(* Logix 5000 project; controller WAGO_765_1504_Sample vendor 1 type 14 code 196 rev 32.14; software revision 32.03 *)

TASK MainTask (continuous, watchdog 500 ms) : MainProgram

MODULES
   Local : vendor 1 type 14 code 196 (5069 0, rev 32.14)
      WAGO_DIO_1504 : vendor 40 type 12 code 1504 (Ethernet 192.168.2.100, rev 1.1, StandardDataDriven RPI 20 ms)
END_MODULES

ADD_ON_INSTRUCTION WAGO_765_1504   (* revision 1.1, vendor WAGO *)
// 765-1504/100-000 AOI, Exclusive Owner Connection Type
// Revision note:
// ModuleConfig.DIO_Process_Data_Layout can be 1 or 0. DO data release is now written to
// Help:
// The WAGO_765_1504 instruction normalizes data received from a WAGO 750-1504/100-000 DIO EIP Adapter. 765-1504/100-000 must be Exclusive Owner (with config).
// This AOI requires ModuleConfig, ModuleInput, and ModuleOutput. These data types are from the EDS file, so do not create these data types--they should already be there if you have the device added.
// ModuleConfig is of type _0028:765_15040100_0000_419E4C60:C:0. This data type allows for configuration of the 765-1504 EIP Adapter.
// ModuleInput is of type _0028:765_15040100_0000_85D36DB4:I:0
// ModuleOutput is of type _0028:765_15040100_0000_AAB94180:O:0
// These data types are from the connection class and should be easily assignable.
// Each port has a pin 2 and pin 4 for input/output data. The DIO configuration is done through the ModuleConfig within the Network Variables. The AOI will break out each pin into individual BOOLs to ease referencing.
// Consult the WAGO 765-1504/100-000 Product Manual for further information about the WAGO I/O System Field DIO EIP Adapter.
VAR_IN_OUT
   ModuleConfig : _0028:765_15040100_0000_419E4C60:C:0; {required}
   ModuleInputs : _0028:765_15040100_0000_85D36DB4:I:0; {required}
   ModuleOutputs : _0028:765_15040100_0000_AAB94180:O:0; {required}
END_VAR
VAR_OUTPUT
   X01_Pin4_Input : BOOL; {access None, visible}
END_VAR
VAR_INPUT
   X01_Pin4_Output : BOOL; {access None, visible}
END_VAR
VAR_OUTPUT
   X01_Pin2_Input : BOOL; {access None, visible}
END_VAR
VAR_INPUT
   X01_Pin2_Output : BOOL; {access None, visible}
END_VAR
VAR_OUTPUT
   X02_Pin4_Input : BOOL; {access None, visible}
END_VAR
VAR_INPUT
   X02_Pin4_Output : BOOL; {access None, visible}
END_VAR
VAR_OUTPUT
   X02_Pin2_Input : BOOL; {access None, visible}
END_VAR
VAR_INPUT
   X02_Pin2_Output : BOOL; {access None, visible}
END_VAR
VAR_OUTPUT
   X03_Pin4_Input : BOOL; {access None, visible}
END_VAR
VAR_INPUT
   X03_Pin4_Output : BOOL; {access None, visible}
END_VAR
VAR_OUTPUT
   X03_Pin2_Input : BOOL; {access None, visible}
END_VAR
VAR_INPUT
   X03_Pin2_Output : BOOL; {access None, visible}
END_VAR
VAR_OUTPUT
   X04_Pin4_Input : BOOL; {access None, visible}
END_VAR
VAR_INPUT
   X04_Pin4_Output : BOOL; {access None, visible}
END_VAR
VAR_OUTPUT
   X04_Pin2_Input : BOOL; {access None, visible}
END_VAR
VAR_INPUT
   X04_Pin2_Output : BOOL; {access None, visible}
END_VAR
VAR
   Step : BOOL; {access None}
END_VAR

ROUTINE Logic   (* ladder *)
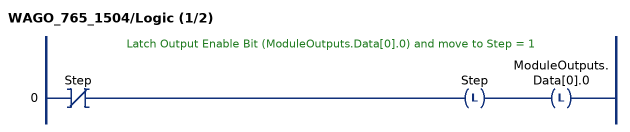
   // Latch Output Enable Bit (ModuleOutputs.Data[0].0) and move to Step = 1
   0: XIO(Step)OTL(Step)OTL(ModuleOutputs.Data[0].0);
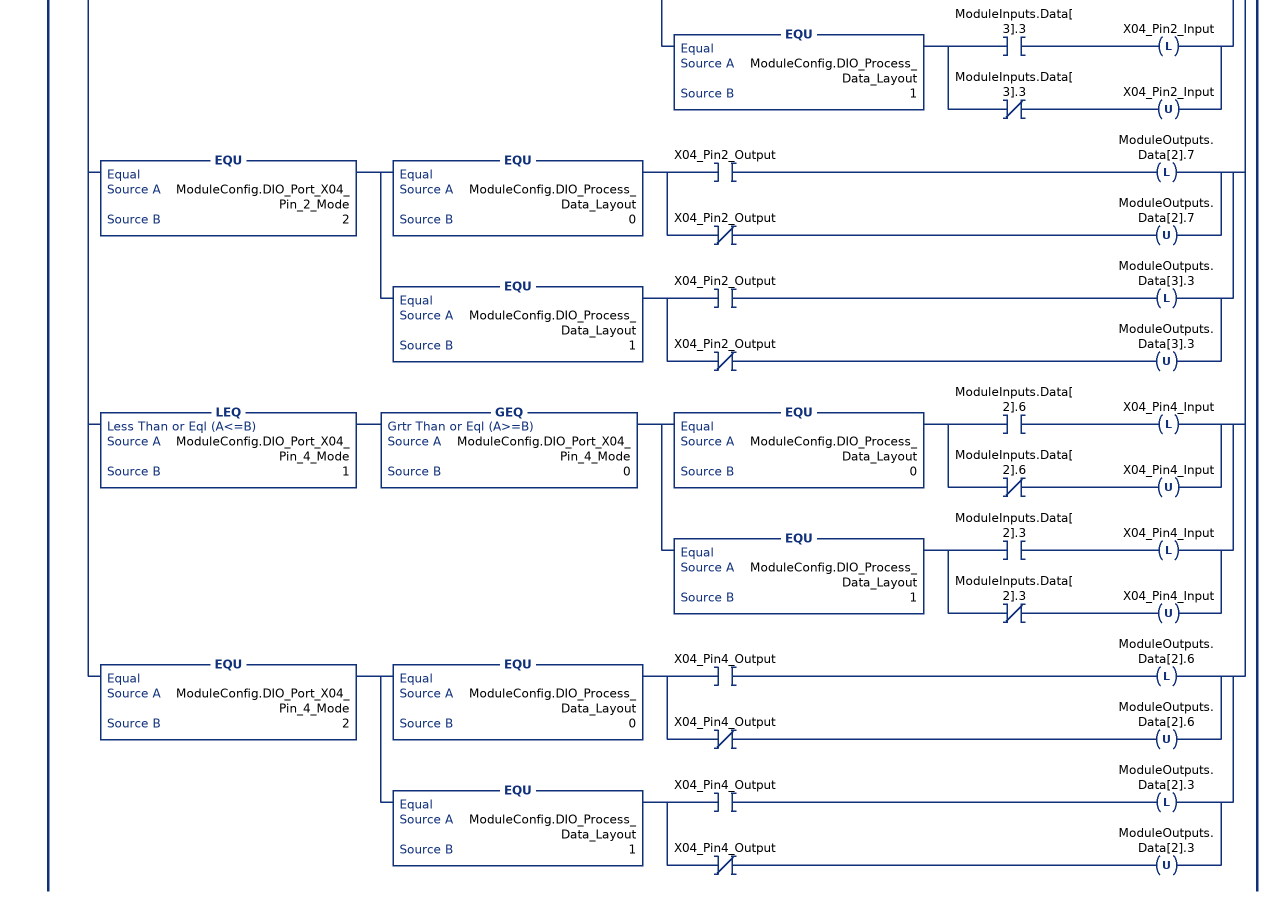
   // Inputs/Outputs read/written are based on ModuleConfig.DIO_Process_Data_Layout.
   1: XIC(Step)[[LEQ(ModuleConfig.DIO_Port_X01_Pin_2_Mode,1) GEQ(ModuleConfig.DIO_Port_X01_Pin_2_Mode,0) [EQU(ModuleConfig.DIO_Process_Data_Layout,0) [XIC(ModuleInputs.Data[2].1) OTL(X01_Pin2_Input) ,XIO(ModuleInputs.Data[2].1) OTU(X01_Pin2_Input) ] ,EQU(ModuleConfig.DIO_Process_Data_Layout,1) [XIC(ModuleInputs.Data[3].0) OTL(X01_Pin2_Input) ,XIO(ModuleInputs.Data[3].0) OTU(X01_Pin2_Input) ] ] ,EQU(ModuleConfig.DIO_Port_X01_Pin_2_Mode,2) [EQU(ModuleConfig.DIO_Process_Data_Layout,0) [XIC(X01_Pin2_Output) OTL(ModuleOutputs.Data[2].1) ,XIO(X01_Pin2_Output) OTU(ModuleOutputs.Data[2].1) ] ,EQU(ModuleConfig.DIO_Process_Data_Layout,1) [XIC(X01_Pin2_Output) OTL(ModuleOutputs.Data[3].0) ,XIO(X01_Pin2_Output) OTU(ModuleOutputs.Data[3].0) ] ] ] ,[LEQ(ModuleConfig.DIO_Port_X01_Pin_4_Mode,1) GEQ(ModuleConfig.DIO_Port_X01_Pin_4_Mode,0) XIC(ModuleInputs.Data[2].0) OTE(X01_Pin4_Input) ,EQU(ModuleConfig.DIO_Port_X01_Pin_4_Mode,2) XIC(X01_Pin4_Output) OTE(ModuleOutputs.Data[2].0) ] ,[LEQ(ModuleConfig.DIO_Port_X02_Pin_2_Mode,1) GEQ(ModuleConfig.DIO_Port_X02_Pin_2_Mode,0) [EQU(ModuleConfig.DIO_Process_Data_Layout,0) [XIC(ModuleInputs.Data[2].3) OTL(X02_Pin2_Input) ,XIO(ModuleInputs.Data[2].3) OTU(X02_Pin2_Input) ] ,EQU(ModuleConfig.DIO_Process_Data_Layout,1) [XIC(ModuleInputs.Data[3].1) OTL(X02_Pin2_Input) ,XIO(ModuleInputs.Data[3].1) OTU(X02_Pin2_Input) ] ] ,EQU(ModuleConfig.DIO_Port_X02_Pin_2_Mode,2) [EQU(ModuleConfig.DIO_Process_Data_Layout,0) [XIC(X02_Pin2_Output) OTL(ModuleOutputs.Data[2].3) ,XIO(X02_Pin2_Output) OTU(ModuleOutputs.Data[2].3) ] ,EQU(ModuleConfig.DIO_Process_Data_Layout,1) [XIC(X02_Pin2_Output) OTL(ModuleOutputs.Data[3].1) ,XIO(X02_Pin2_Output) OTU(ModuleOutputs.Data[3].1) ] ] ] ,[LEQ(ModuleConfig.DIO_Port_X02_Pin_4_Mode,1) GEQ(ModuleConfig.DIO_Port_X02_Pin_4_Mode,0) [EQU(ModuleConfig.DIO_Process_Data_Layout,0) [XIC(ModuleInputs.Data[2].2) OTL(X02_Pin4_Input) ,XIO(ModuleInputs.Data[2].2) OTU(X02_Pin4_Input) ] ,EQU(ModuleConfig.DIO_Process_Data_Layout,1) [XIC(ModuleInputs.Data[2].1) OTL(X02_Pin4_Input) ,XIO(ModuleInputs.Data[2].1) OTU(X02_Pin4_Input) ] ] ,EQU(ModuleConfig.DIO_Port_X02_Pin_4_Mode,2) [EQU(ModuleConfig.DIO_Process_Data_Layout,0) [XIC(X02_Pin4_Output) OTL(ModuleOutputs.Data[2].2) ,XIO(X02_Pin4_Output) OTU(ModuleOutputs.Data[2].2) ] ,EQU(ModuleConfig.DIO_Process_Data_Layout,1) [XIC(X02_Pin4_Output) OTL(ModuleOutputs.Data[2].1) ,XIO(X02_Pin4_Output) OTU(ModuleOutputs.Data[2].1) ] ] ] ,[LEQ(ModuleConfig.DIO_Port_X03_Pin_2_Mode,1) GEQ(ModuleConfig.DIO_Port_X03_Pin_2_Mode,0) [EQU(ModuleConfig.DIO_Process_Data_Layout,0) [XIC(ModuleInputs.Data[2].5) OTL(X03_Pin2_Input) ,XIO(ModuleInputs.Data[2].5) OTU(X03_Pin2_Input) ] ,EQU(ModuleConfig.DIO_Process_Data_Layout,1) [XIC(ModuleInputs.Data[3].2) OTL(X03_Pin2_Input) ,XIO(ModuleInputs.Data[3].2) OTU(X03_Pin2_Input) ] ] ,EQU(ModuleConfig.DIO_Port_X03_Pin_2_Mode,2) [EQU(ModuleConfig.DIO_Process_Data_Layout,0) [XIC(X03_Pin2_Output) OTL(ModuleOutputs.Data[2].5) ,XIO(X03_Pin2_Output) OTU(ModuleOutputs.Data[2].5) ] ,EQU(ModuleConfig.DIO_Process_Data_Layout,1) [XIC(X03_Pin2_Output) OTL(ModuleOutputs.Data[3].2) ,XIO(X03_Pin2_Output) OTU(ModuleOutputs.Data[3].2) ] ] ] ,[LEQ(ModuleConfig.DIO_Port_X03_Pin_4_Mode,1) GEQ(ModuleConfig.DIO_Port_X03_Pin_4_Mode,0) [EQU(ModuleConfig.DIO_Process_Data_Layout,0) [XIC(ModuleInputs.Data[2].4) OTL(X03_Pin4_Input) ,XIO(ModuleInputs.Data[2].4) OTU(X03_Pin4_Input) ] ,EQU(ModuleConfig.DIO_Process_Data_Layout,1) [XIC(ModuleInputs.Data[2].2) OTL(X03_Pin4_Input) ,XIO(ModuleInputs.Data[2].2) OTU(X03_Pin4_Input) ] ] ,EQU(ModuleConfig.DIO_Port_X03_Pin_4_Mode,2) [EQU(ModuleConfig.DIO_Process_Data_Layout,0) [XIC(X03_Pin4_Output) OTL(ModuleOutputs.Data[2].4) ,XIO(X03_Pin4_Output) OTU(ModuleOutputs.Data[2].4) ] ,EQU(ModuleConfig.DIO_Process_Data_Layout,1) [XIC(X03_Pin4_Output) OTL(ModuleOutputs.Data[2].2) ,XIO(X03_Pin4_Output) OTU(ModuleOutputs.Data[2].2) ] ] ] ,[LEQ(ModuleConfig.DIO_Port_X04_Pin_2_Mode,1) GEQ(ModuleConfig.DIO_Port_X04_Pin_2_Mode,0) [EQU(ModuleConfig.DIO_Process_Data_Layout,0) [XIC(ModuleInputs.Data[2].7) OTL(X04_Pin2_Input) ,XIO(ModuleInputs.Data[2].7) OTU(X04_Pin2_Input) ] ,EQU(ModuleConfig.DIO_Process_Data_Layout,1) [XIC(ModuleInputs.Data[3].3) OTL(X04_Pin2_Input) ,XIO(ModuleInputs.Data[3].3) OTU(X04_Pin2_Input) ] ] ,EQU(ModuleConfig.DIO_Port_X04_Pin_2_Mode,2) [EQU(ModuleConfig.DIO_Process_Data_Layout,0) [XIC(X04_Pin2_Output) OTL(ModuleOutputs.Data[2].7) ,XIO(X04_Pin2_Output) OTU(ModuleOutputs.Data[2].7) ] ,EQU(ModuleConfig.DIO_Process_Data_Layout,1) [XIC(X04_Pin2_Output) OTL(ModuleOutputs.Data[3].3) ,XIO(X04_Pin2_Output) OTU(ModuleOutputs.Data[3].3) ] ] ] ,[LEQ(ModuleConfig.DIO_Port_X04_Pin_4_Mode,1) GEQ(ModuleConfig.DIO_Port_X04_Pin_4_Mode,0) [EQU(ModuleConfig.DIO_Process_Data_Layout,0) [XIC(ModuleInputs.Data[2].6) OTL(X04_Pin4_Input) ,XIO(ModuleInputs.Data[2].6) OTU(X04_Pin4_Input) ] ,EQU(ModuleConfig.DIO_Process_Data_Layout,1) [XIC(ModuleInputs.Data[2].3) OTL(X04_Pin4_Input) ,XIO(ModuleInputs.Data[2].3) OTU(X04_Pin4_Input) ] ] ,EQU(ModuleConfig.DIO_Port_X04_Pin_4_Mode,2) [EQU(ModuleConfig.DIO_Process_Data_Layout,0) [XIC(X04_Pin4_Output) OTL(ModuleOutputs.Data[2].6) ,XIO(X04_Pin4_Output) OTU(ModuleOutputs.Data[2].6) ] ,EQU(ModuleConfig.DIO_Process_Data_Layout,1) [XIC(X04_Pin4_Output) OTL(ModuleOutputs.Data[2].3) ,XIO(X04_Pin4_Output) OTU(ModuleOutputs.Data[2].3) ] ] ] ];
END_ROUTINE
END_ADD_ON_INSTRUCTION

VAR_GLOBAL   (* controller tags *)
   Fail_Safe_Config : DINT[16];   // 0 = Low on loss of communication 1 = High on Loss of communication 2 = Maintain last known value
   Filter_Config : DINT[16];   // 0 = No Filter 1 = 1 microsecond 2 = 10 microsecond 3 = 100 microsecond 4 = 1 millisecond 5 = 2 millisecond 6 = 3 millisecond
   my_1504 : WAGO_765_1504;
   zzz_Wago_Flag : DINT;   // WAGO IO Test Bits
END_VAR

PROGRAM MainProgram   (* main routine MainRoutine *)

ROUTINE MainRoutine   (* ladder *)
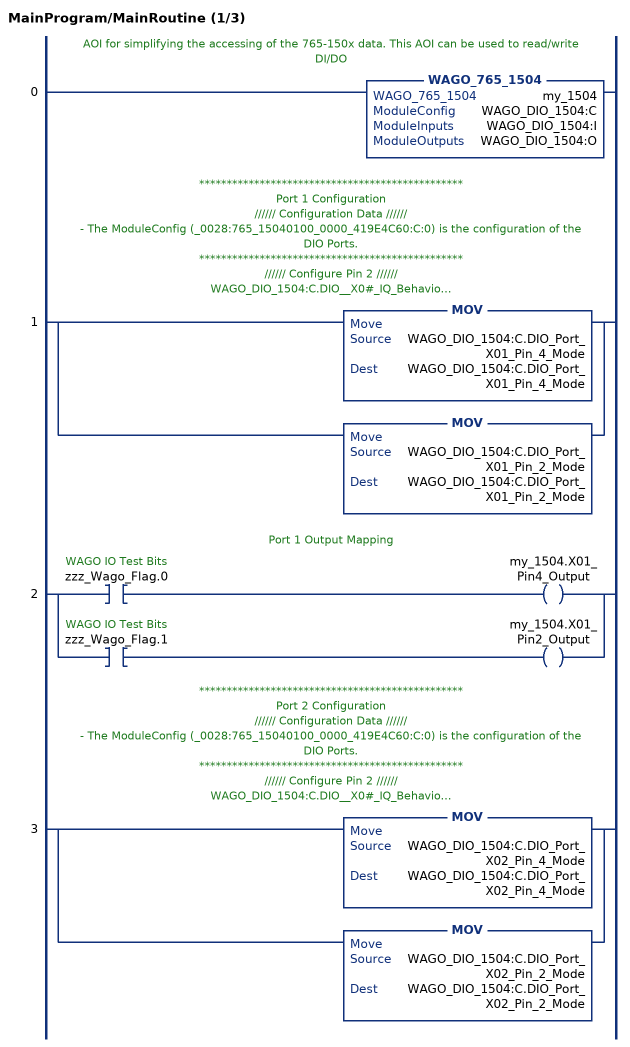
   // AOI for simplifying the accessing of the 765-150x data. This AOI can be used to read/write DI/DO
   0: WAGO_765_1504(my_1504,WAGO_DIO_1504:C,WAGO_DIO_1504:I,WAGO_DIO_1504:O);
   // ************************************************
   // Port 1 Configuration
   // ////// Configuration Data //////
   //       - The ModuleConfig (_0028:765_15040100_0000_419E4C60:C:0) is the configuration of the DIO Ports.
   // ************************************************
   // ////// Configure Pin 2 //////
   // WAGO_DIO_1504:C.DIO__X0#_IQ_Behavior
   // (0 = disabled, 1 = DI, 2 = DO)
   // ////// Configure Pin 4 //////
   // WAGO_DIO_1504:C.DIO_Port_X0#_Port_Mode
   // (0 = disabled, 1 = DI, 2 = DO)
   1: [MOV(WAGO_DIO_1504:C.DIO_Port_X01_Pin_4_Mode,WAGO_DIO_1504:C.DIO_Port_X01_Pin_4_Mode) ,MOV(WAGO_DIO_1504:C.DIO_Port_X01_Pin_2_Mode,WAGO_DIO_1504:C.DIO_Port_X01_Pin_2_Mode) ];
   // Port 1 Output Mapping
   2: [XIC(zzz_Wago_Flag.0) OTE(my_1504.X01_Pin4_Output) ,XIC(zzz_Wago_Flag.1) OTE(my_1504.X01_Pin2_Output) ];
   // ************************************************
   // Port 2 Configuration
   // ////// Configuration Data //////
   //       - The ModuleConfig (_0028:765_15040100_0000_419E4C60:C:0) is the configuration of the DIO Ports.
   // ************************************************
   // ////// Configure Pin 2 //////
   // WAGO_DIO_1504:C.DIO__X0#_IQ_Behavior
   // (0 = disabled, 1 = DI, 2 = DO)
   // ////// Configure Pin 4 //////
   // WAGO_DIO_1504:C.DIO_Port_X0#_Port_Mode
   // (0 = disabled, 1 = DI, 2 = DO)
   3: [MOV(WAGO_DIO_1504:C.DIO_Port_X02_Pin_4_Mode,WAGO_DIO_1504:C.DIO_Port_X02_Pin_4_Mode) ,MOV(WAGO_DIO_1504:C.DIO_Port_X02_Pin_2_Mode,WAGO_DIO_1504:C.DIO_Port_X02_Pin_2_Mode) ];
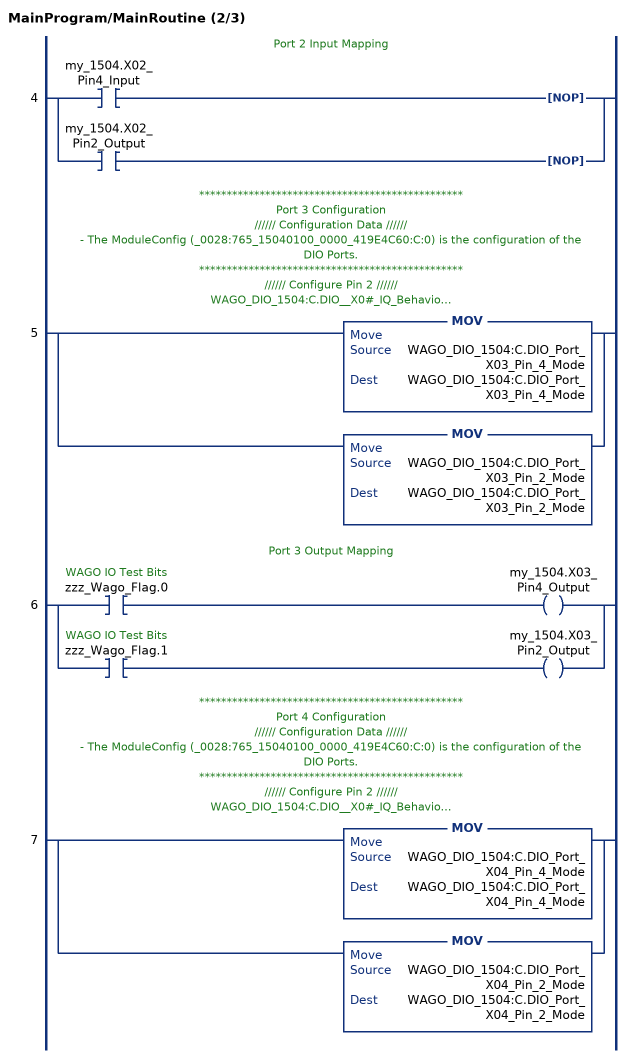
   // Port 2 Input Mapping
   4: [XIC(my_1504.X02_Pin4_Input) NOP() ,XIC(my_1504.X02_Pin2_Output) NOP() ];
   // ************************************************
   // Port 3 Configuration
   // ////// Configuration Data //////
   //       - The ModuleConfig (_0028:765_15040100_0000_419E4C60:C:0) is the configuration of the DIO Ports.
   // ************************************************
   // ////// Configure Pin 2 //////
   // WAGO_DIO_1504:C.DIO__X0#_IQ_Behavior
   // (0 = disabled, 1 = DI, 2 = DO)
   // ////// Configure Pin 4 //////
   // WAGO_DIO_1504:C.DIO_Port_X0#_Port_Mode
   // (0 = disabled, 1 = DI, 2 = DO)
   5: [MOV(WAGO_DIO_1504:C.DIO_Port_X03_Pin_4_Mode,WAGO_DIO_1504:C.DIO_Port_X03_Pin_4_Mode) ,MOV(WAGO_DIO_1504:C.DIO_Port_X03_Pin_2_Mode,WAGO_DIO_1504:C.DIO_Port_X03_Pin_2_Mode) ];
   // Port 3 Output Mapping
   6: [XIC(zzz_Wago_Flag.0) OTE(my_1504.X03_Pin4_Output) ,XIC(zzz_Wago_Flag.1) OTE(my_1504.X03_Pin2_Output) ];
   // ************************************************
   // Port 4 Configuration
   // ////// Configuration Data //////
   //       - The ModuleConfig (_0028:765_15040100_0000_419E4C60:C:0) is the configuration of the DIO Ports.
   // ************************************************
   // ////// Configure Pin 2 //////
   // WAGO_DIO_1504:C.DIO__X0#_IQ_Behavior
   // (0 = disabled, 1 = DI, 2 = DO)
   // ////// Configure Pin 4 //////
   // WAGO_DIO_1504:C.DIO_Port_X0#_Port_Mode
   // (0 = disabled, 1 = DI, 2 = DO)
   7: [MOV(WAGO_DIO_1504:C.DIO_Port_X04_Pin_4_Mode,WAGO_DIO_1504:C.DIO_Port_X04_Pin_4_Mode) ,MOV(WAGO_DIO_1504:C.DIO_Port_X04_Pin_2_Mode,WAGO_DIO_1504:C.DIO_Port_X04_Pin_2_Mode) ];
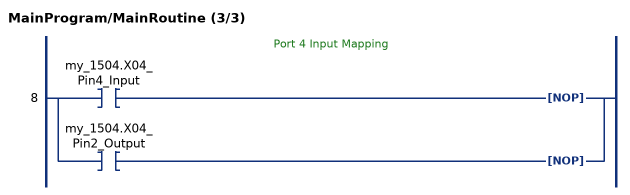
   // Port 4 Input Mapping
   8: [XIC(my_1504.X04_Pin4_Input) NOP() ,XIC(my_1504.X04_Pin2_Output) NOP() ];
END_ROUTINE
END_PROGRAM
